TYPE GearInPos_Statuses_typ :
	STRUCT
		StartSync       : BOOL;
        InSync          : BOOL;
        CommandAborted  : BOOL;
		Active 			: BOOL;
		Busy			: BOOL;

	END_STRUCT
END_TYPE

(* stored: Version 1.1.0.1, ProductVersion 3.1.4024.3
   DUT GearInPos_Statuses_typ: Id {e87a595e-402a-0ff2-235d-8de945d9cb25} *)
